PROGRAM MAIN
VAR
	bIsStartPressed : BOOL;
	bIsStopPressed : BOOL;
	bIsBlinkPressed : BOOL;

	fbTrafficLight : FB_TrafficLight;
	
	dwRedTimeOn : DWORD := 8000;
	
	dwRedAndYellowTimeOn : DWORD := 1000;
	
	dwGreenTimeOn : DWORD := 5000;
	
	dwGreenBlinkingDuration : DWORD := 2000;
	dwGreenBlinkingTimeOn : DWORD := 250;
	dwGreenBlinkingTimeOff : DWORD := 100;
	
	dwYellowTimeOn : DWORD := 1000;
	
	dwYellowBlinkingTimeOn : DWORD := 250;
	dwYellowBlinkingTimeOff : DWORD := 100;
END_VAR

fbTrafficLight(bIsStartPressed := bIsStartPressed, bIsStopPressed := bIsStopPressed, bIsBlinkPressed := bIsBlinkPressed,
			   dwRedTimeOn := dwRedTimeOn,
			   dwRedAndYellowTimeOn := dwRedAndYellowTimeOn, 
			   dwGreenTimeOn := dwGreenTimeOn,
			   dwGreenBlinkingDuration := dwGreenBlinkingDuration, dwGreenBlinkingTimeOn := dwGreenBlinkingTimeOn, dwGreenBlinkingTimeOff := dwGreenBlinkingTimeOff,
			   dwYellowTimeOn := dwYellowTimeOn,
			   dwYellowBlinkingTimeOn := dwYellowBlinkingTimeOn, dwYellowBlinkingTimeOff := dwYellowBlinkingTimeOff,);		   
			   
//// For connection with hardware
//fbTrafficLight(dwRedTimeOn := dwRedTimeOn,
//			   dwRedAndYellowTimeOn := dwRedAndYellowTimeOn, 
//			   dwGreenTimeOn := dwGreenTimeOn,
//			   dwGreenBlinkingDuration := dwGreenBlinkingDuration, dwGreenBlinkingTimeOn := dwGreenBlinkingTimeOn, dwGreenBlinkingTimeOff := dwGreenBlinkingTimeOff,
//			   dwYellowTimeOn := dwYellowTimeOn,
//			   dwYellowBlinkingTimeOn := dwYellowBlinkingTimeOn, dwYellowBlinkingTimeOff := dwYellowBlinkingTimeOff,);

END_PROGRAM

(* stored: Version 1.1.0.1, ProductVersion 3.1.4024.12
   POU MAIN: Id {de73dcfc-be11-4121-8cb0-5c8df10a409c}, SpecialFunc None *)
